FUNCTION_BLOCK T_ConnectionTCPIP EXTENDS T_NamedBase IMPLEMENTS I_Connection
VAR
	connection : T_TcpClientConnection;
	sender : T_TcpSend;
	receiver : T_TcpRecieve;
	init : BOOL;
	state : (IDLE, WORKING);
  
  IsConnectedTrigger : R_TRIG;
  IsNotConnectedTrigger : F_TRIG;
END_VAR

METHOD Connect 
VAR_INPUT
  ip : T_IPv4Addr;
  port : UINT;
  timeout : TIME;
END_VAR
connection.Connect(ip, port, timeout);
LogInfo('Connecting');
END_METHOD

METHOD PUBLIC CyclicLogic
VAR_INST
  trigConnected : R_TRIG;
  isNotConnectedTrigger : F_TRIG;
  trigErrReceive : R_TRIG;
END_VAR
IF NOT init THEN
	init := TRUE;
END_IF

connection.CyclicLogic();
trigConnected(CLK := connection.IsConnected);

IF trigConnected.Q THEN
	sender.SetSocket(connection.Socket);
	receiver.SetSocket(connection.Socket);
  receiver.Start();
	LogDebug('Connected - setting socket on sender and receiver.');
END_IF

isNotConnectedTrigger(CLK := connection.IsConnected);
IF isNotConnectedTrigger.Q THEN
  receiver.Stop();
END_IF

IF NOT connection.IsConnected THEN
 	RETURN;
END_IF

sender.CyclicLogic();
receiver.CyclicLogic();

// If error detected on receive, need to try disconnecting and reconnecting
trigErrReceive(CLK:= IsErrorReceive, Q=> );
IF trigErrReceive.Q THEN
	ErrorReceive();
END_IF
END_METHOD

METHOD Disconnect
connection.Disconnect();
LogInfo('Disconnecting');
END_METHOD

PROPERTY ErrID : UDINT
GET
IF IsErrorConnect THEN
	ErrID := connection.ErrID;
ELSIF IsErrorSend THEN
	ErrID := sender.ErrID;
ELSIF IsErrorReceive THEN
	ErrID := receiver.ErrID;
END_IF
END_GET
END_PROPERTY

METHOD ErrorReceive : BOOL
LogError('Receive Error');
Disconnect();
END_METHOD

PROPERTY IsBusy : BOOL
GET
IsBusy := connection.IsBusy OR sender.IsBusy OR receiver.IsBusy;
END_GET
END_PROPERTY

PROPERTY IsConnected : BOOL
GET
IsConnected := connection.IsConnected;
END_GET
END_PROPERTY

PROPERTY IsErrorConnect : Bool
GET
IsErrorConnect := connection.IsError;
END_GET
END_PROPERTY

PROPERTY IsErrorReceive : BOOL
GET
IsErrorReceive := receiver.IsError;
END_GET
END_PROPERTY

PROPERTY IsErrorSend : BOOL
GET
IsErrorSend := sender.IsError;
END_GET
END_PROPERTY

METHOD Receive : BOOL // TRUE if new data recieved.
VAR_OUTPUT 
  data : ARRAY [1..RoboConnectParams.receiveBufferSize] OF BYTE;  // Contents of received buffer
  receiveLength : UDINT; // length of data received.
END_VAR
IF NOT connection.IsConnected THEN
  LogWarning('Cannot receive message, NOT connected');
  RETURN;
END_IF

Receive :=
  receiver.TryGetBuffer(
    result := data,
    receiveLength => receiveLength
  );
END_METHOD

METHOD Send : BOOL
VAR_INPUT
  message : T_Maxstring;
END_VAR
IF NOT connection.IsConnected THEN
  LogWarning('Cannot send message, not connected');
  RETURN;
END_IF

LogInfo(CONCAT('Sending message : ', message));
sender.Send(message);
Send := TRUE;
END_METHOD

PROPERTY PUBLIC SendDone : BOOL
GET
SendDone := NOT sender.IsBusy;
END_GET
END_PROPERTY

END_FUNCTION_BLOCK

(* stored: Version 1.1.0.1
   POU T_ConnectionTCPIP: Id {dfdbd582-0c2f-4b59-80e4-5d84cd3715d5}, SpecialFunc None
   Folder Methods: Id {b246d1b9-d86b-4dee-bfb8-bf8852170adb}
   Folder Properties: Id {696d23c4-bfc5-410e-92c8-70d9c2387824}
   Method Connect: Id {6fff02a0-134e-46fe-b8e6-d7dc6171bd6d}
   Method CyclicLogic: Id {132d8014-9794-4a0e-9813-c917f683b470}
   Method Disconnect: Id {e1f68167-2fb7-4bed-a2f7-bf27332b2011}
   Property ErrID: Id {edc96c3d-f9ae-4be2-8ecb-49f7931b19d8}
   Get Get: Id {f75277bf-1f24-4abb-8eb1-b92635661e31}
   Method ErrorReceive: Id {de667186-f63c-40e2-b4f3-1a0025d7746d}
   Property IsBusy: Id {748064e5-625d-4fe8-9c92-4e7d7d234f20}
   Get Get: Id {c453cbda-0252-4943-9bc9-921ab58fcb3d}
   Property IsConnected: Id {cb8b73ce-4a0d-4feb-93d2-345ebecad54d}
   Get Get: Id {18778902-73d1-4ef8-b294-a4fce202d8d2}
   Property IsErrorConnect: Id {4acd44be-5275-467a-8eec-18fa71242114}
   Get Get: Id {691fca2f-6e91-4dda-89b1-e1ce595141cc}
   Property IsErrorReceive: Id {2abadd84-c77d-49f9-8282-91c3f7c5d809}
   Get Get: Id {24a43233-15d0-4a10-bcef-e40482d684a8}
   Property IsErrorSend: Id {7aa0ba27-18a4-4e50-ac57-e4020055c376}
   Get Get: Id {8729f01d-e697-4063-ba7a-8e643d083f15}
   Method Receive: Id {2413eb5d-c13b-4da5-b312-face6dde8e72}
   Method Send: Id {69776a4d-48a5-44be-95ec-4125eb36f784}
   Property SendDone: Id {67e5ce5b-36fc-4956-a2c0-0f36eb74b48d}
   Get Get: Id {cb081cc7-2675-447a-97b3-d76e545704d9} *)
